TYPE "LubrValve_Config"
VERSION : 0.1
// Block: LubrValve_Config
   STRUCT
      WorkMode : Int;
      CounterMode : Int;
      ValveType : Int;
      ManualCmdTimeOut : Time;
   END_STRUCT;

END_TYPE
